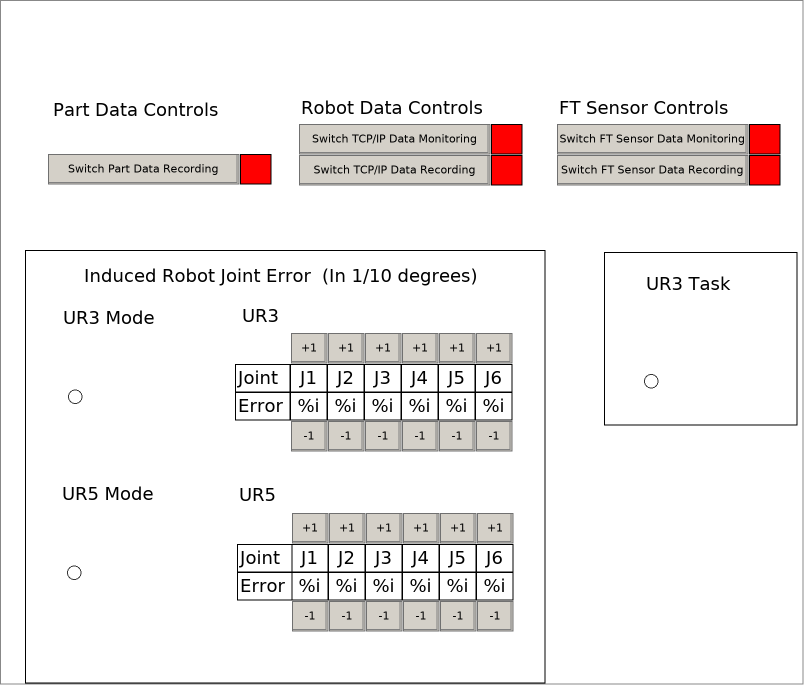
VISUALIZATION Settings  // 804x685
    RoundedRectangle (604,252 193x173)
    RoundedRectangle (25,250 520x433)
    Button (299,124 191x30), "Switch TCP/IP Data Monitoring"
        OnMouseClick: toggle Global.bActivateTCPIPDataCollection
    Button (299,155 191x30), "Switch TCP/IP Data Recording"
        OnMouseClick: toggle Global.bActivateTCPIPDataRecording
    Rectangle (491,124 31x30), colour toggle: Global.bActivateTCPIPDataCollection
    Rectangle (491,155 31x30), colour toggle: Global.bActivateTCPIPDataRecording
    Label (298,93 246x30), "Robot Data Controls"
    Label (81,261 507x30), "Induced Robot Joint Error (In 1/10 degrees)"
    Label (239,301 77x30), "UR3"
    Label (236,480 77x30), "UR5"
    Rectangle (291,572 37x28), "%i", text variable: Global.stUR5.InducedJointError[1]
    Button (292,513 36x30), "+1"
        OnMouseClick: execute { Global.stUR5.InducedJointError[1] := Global.stUR5.InducedJointError[1] + 1; }
    Button (292,601 36x30), "-1"
        OnMouseClick: execute { Global.stUR5.InducedJointError[1] := Global.stUR5.InducedJointError[1] - 1; }
    Rectangle (291,544 37x28), "J1"
    Rectangle (328,572 37x28), "%i", text variable: Global.stUR5.InducedJointError[2]
    Button (329,513 36x30), "+1"
        OnMouseClick: execute { Global.stUR5.InducedJointError[2] := Global.stUR5.InducedJointError[2] + 1; }
    Button (329,601 36x30), "-1"
        OnMouseClick: execute { Global.stUR5.InducedJointError[2] := Global.stUR5.InducedJointError[2] - 1; }
    Rectangle (328,544 37x28), "J2"
    Rectangle (365,572 37x28), "%i", text variable: Global.stUR5.InducedJointError[3]
    Button (366,513 36x30), "+1"
        OnMouseClick: execute { Global.stUR5.InducedJointError[3] := Global.stUR5.InducedJointError[3] + 1; }
    Button (366,601 36x30), "-1"
        OnMouseClick: execute { Global.stUR5.InducedJointError[3] := Global.stUR5.InducedJointError[3] - 1; }
    Rectangle (365,544 37x28), "J3"
    Rectangle (402,572 37x28), "%i", text variable: Global.stUR5.InducedJointError[4]
    Button (403,513 36x30), "+1"
        OnMouseClick: execute { Global.stUR5.InducedJointError[4] := Global.stUR5.InducedJointError[4] + 1; }
    Button (403,601 36x30), "-1"
        OnMouseClick: execute { Global.stUR5.InducedJointError[4] := Global.stUR5.InducedJointError[4] - 1; }
    Rectangle (402,544 37x28), "J4"
    Rectangle (439,572 37x28), "%i", text variable: Global.stUR5.InducedJointError[5]
    Button (440,513 36x30), "+1"
        OnMouseClick: execute { Global.stUR5.InducedJointError[5] := Global.stUR5.InducedJointError[5] + 1; }
    Button (440,601 36x30), "-1"
        OnMouseClick: execute { Global.stUR5.InducedJointError[5] := Global.stUR5.InducedJointError[5] - 1; }
    Rectangle (439,544 37x28), "J5"
    Rectangle (476,572 37x28), "%i", text variable: Global.stUR5.InducedJointError[6]
    Button (477,513 36x30), "+1"
        OnMouseClick: execute { Global.stUR5.InducedJointError[6] := Global.stUR5.InducedJointError[6] + 1; }
    Button (477,601 36x30), "-1"
        OnMouseClick: execute { Global.stUR5.InducedJointError[6] := Global.stUR5.InducedJointError[6] - 1; }
    Rectangle (476,544 37x28), "J6"
    Rectangle (237,544 55x28), "Joint"
    Rectangle (237,572 55x28), "Error", text variable: Global.stUR5.InducedJointError[1]
    Rectangle (290,392 37x28), "%i", text variable: Global.stUR3.InducedJointError[1]
    Button (291,333 36x30), "+1"
        OnMouseClick: execute { Global.stUR3.InducedJointError[1] := Global.stUR3.InducedJointError[1] + 1; }
    Button (291,421 36x30), "-1"
        OnMouseClick: execute { Global.stUR3.InducedJointError[1] := Global.stUR3.InducedJointError[1] - 1; }
    Rectangle (290,364 37x28), "J1"
    Rectangle (327,392 37x28), "%i", text variable: Global.stUR3.InducedJointError[2]
    Button (328,333 36x30), "+1"
        OnMouseClick: execute { Global.stUR3.InducedJointError[2] := Global.stUR3.InducedJointError[2] + 1; }
    Button (328,421 36x30), "-1"
        OnMouseClick: execute { Global.stUR3.InducedJointError[2] := Global.stUR3.InducedJointError[2] - 1; }
    Rectangle (327,364 37x28), "J2"
    Rectangle (364,392 37x28), "%i", text variable: Global.stUR3.InducedJointError[3]
    Button (365,333 36x30), "+1"
        OnMouseClick: execute { Global.stUR3.InducedJointError[3] := Global.stUR3.InducedJointError[3] + 1; }
    Button (365,421 36x30), "-1"
        OnMouseClick: execute { Global.stUR3.InducedJointError[3] := Global.stUR3.InducedJointError[3] - 1; }
    Rectangle (364,364 37x28), "J3"
    Rectangle (401,392 37x28), "%i", text variable: Global.stUR3.InducedJointError[4]
    Button (402,333 36x30), "+1"
        OnMouseClick: execute { Global.stUR3.InducedJointError[4] := Global.stUR3.InducedJointError[4] + 1; }
    Button (402,421 36x30), "-1"
        OnMouseClick: execute { Global.stUR3.InducedJointError[4] := Global.stUR3.InducedJointError[4] - 1; }
    Rectangle (401,364 37x28), "J4"
    Rectangle (438,392 37x28), "%i", text variable: Global.stUR3.InducedJointError[5]
    Button (439,333 36x30), "+1"
        OnMouseClick: execute { Global.stUR3.InducedJointError[5] := Global.stUR3.InducedJointError[5] + 1; }
    Button (439,421 36x30), "-1"
        OnMouseClick: execute { Global.stUR3.InducedJointError[5] := Global.stUR3.InducedJointError[5] - 1; }
    Rectangle (438,364 37x28), "J5"
    Rectangle (475,392 37x28), "%i", text variable: Global.stUR3.InducedJointError[6]
    Button (476,333 36x30), "+1"
        OnMouseClick: execute { Global.stUR3.InducedJointError[6] := Global.stUR3.InducedJointError[6] + 1; }
    Button (476,421 36x30), "-1"
        OnMouseClick: execute { Global.stUR3.InducedJointError[6] := Global.stUR3.InducedJointError[6] - 1; }
    Rectangle (475,364 37x28), "J6"
    Rectangle (235,364 55x28), "Joint"
    Rectangle (235,392 55x28), "Error", text variable: Global.stUR5.InducedJointError[1]
    Button (557,124 191x30), "Switch FT Sensor Data Monitoring"
        OnMouseClick: toggle Global.bActivateFTDataCollection
    Button (557,155 191x30), "Switch FT Sensor Data Recording"
        OnMouseClick: toggle Global.bActivateFTDataRecording
    Rectangle (749,124 31x30), colour toggle: Global.bActivateFTDataCollection
    Rectangle (749,155 31x30), colour toggle: Global.bActivateFTDataRecording
    Label (556,93 246x30), "FT Sensor Controls"
    Button (48,154 191x30), "Switch Part Data Recording"
        OnMouseClick: toggle Global.bActivatePartDataRecording
    Rectangle (240,154 31x30), colour toggle: Global.bActivatePartDataRecording
    Label (50,95 246x30), "Part Data Controls"
    RadioButton (66,350 150x93), variable: Global.stUR3.InducedJErrorType
        Areas[0]: Text=Off
        Areas[1]: Text=Encoder Slip
        Areas[2]: Text=Backlash
    Label (60,303 147x30), "UR3 Mode"
    RadioButton (65,526 150x93), variable: Global.stUR5.InducedJErrorType
        Areas[0]: Text=Off
        Areas[1]: Text=Encoder Slip
        Areas[2]: Text=Backlash
    Label (59,479 147x30), "UR5 Mode"
    RadioButton (642,306 150x150), variable: Global.nActiveUR3Task
        Areas[0]: Text=Box and Circle
        Areas[1]: Text=NIST Logo
        Areas[2]: Text=Reserved
    Label (643,269 103x30), "UR3 Task"
END_VISUALIZATION

(* stored: Version 1.1.0.1, ProductVersion 3.1.4020.12
   Visu Settings: Id {93f14146-749e-4200-b05e-0f387fa03c7b} *)
